// TIA Portal V19 export
TYPE "LEXCHANGETRAY_typeConstraintRollerEm_toHandlingXyzFeedback"
// stored: Access Published
   STRUCT
      catchEnable : Bool;   // 允许抓取
   END_STRUCT;
END_TYPE
